FUNCTION_BLOCK Q_ChangePolygonPoint (* Command Change Polygon Point( Part 6 - F.52 ) *)
  (* Standard: ISO 11783-6; Description: Copyright (c) 2022 HR Agrartechnik GmbH This program and the accompanying materials are made available under the terms of the Eclipse Public License 2.0 which is available at https://www.eclipse.org/legal/epl-2.0/ SPDX-License-Identifier: EPL-2.0 see Description Tab *)
  (* Version 1.0, 2022-07-08, Franz Höpfinger, HR Agrartechnik GmbH *)
  PACKAGE isobus::UT::Q;
  IMPORT eclipse4diac::core::TypeHash;
  IMPORT isobus::UT::Q::IDs::ID_NULL;
  (* Documentation:
  Command Change Polygon Point( Part 6 - F.52 )
   This command is used by a Working Set to modify a point in an Output Polygon object.
   param[in] {objectID, uint16_t}
   Object ID of the Output Polygon object to change
   param[in] {pointIndex, uint8_t}
   Point index of the point to replace.
   param[in] {newXValue, uint16_t}
   New X value of a point relative to the top left corner of the polygon
   param[in] {newYValue, uint16_t}
   New Y value of a point relative to the top left corner of the polygon
   Return Values: 
   int16_t
    - VT_E_NO_ERR (0) - OK
   - VT_E_OVERFLOW (-6) - buffer overflow
   - VT_E_NOACT (-8) - Command not possible in current state
   - VT_E_NO_INSTANCE (-21) - No VT client available
   - VT_E_ISO_INSTANCE_INVALID (-129) - Identifier for instance (connection) invalid
   - VT_E_NOT_ALIVE (-130) - Identifier for instance valid, but VT Dead.
  *)
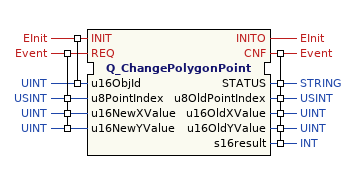
  EVENT_INPUT
    INIT : EInit WITH u16ObjId; (* Service Initialization *)
    REQ WITH u8PointIndex, u16NewXValue, u16NewYValue; (* Service Request *)
  END_EVENT
  EVENT_OUTPUT
    INITO : EInit; (* Initialization Confirm *)
    CNF WITH STATUS, s16result, u8OldPointIndex, u16OldXValue, u16OldYValue; (* Confirmation of Requested Service *)
  END_EVENT
  VAR_INPUT
    u16ObjId : UINT := ID_NULL; (* Object ID of the Output Polygon object to change *)
    u8PointIndex : USINT; (* Point index of the point to replace. *)
    u16NewXValue : UINT; (* New X value of a point relative to the top left corner of the polygon *)
    u16NewYValue : UINT; (* New Y value of a point relative to the top left corner of the polygon *)
  END_VAR
  VAR_OUTPUT
    STATUS : STRING; (* Service Status *)
    u8OldPointIndex : USINT; (* Old point index of the point to replace. *)
    u16OldXValue : UINT; (* Old X value of a point relative to the top left corner of the polygon *)
    u16OldYValue : UINT; (* Old Y value of a point relative to the top left corner of the polygon *)
    s16result : INT; (* retval see description *)
  END_VAR
END_FUNCTION_BLOCK
